// TIA Portal V17 export
// export: Created 2025-06-26T06:49:24.3780906Z, ExportSetting WithDefaults, DisplayName Totally Integrated Automation Portal, DisplayVersion V17 Update 8, DisplayName TIA Portal Openness, DisplayVersion V17 Update 8, DisplayName TIA Portal Version Control Interface, DisplayVersion V17, DisplayName STEP 7 Professional, DisplayVersion V17 Update 8, DisplayName STEP 7 Safety, DisplayVersion V17 Update 6, DisplayName WinCC Advanced, DisplayVersion V17 Update 8
DATA_BLOCK "HMI-Communication_DB"   // DB3
VERSION : 0.1
// stored: AutoNumber true, DBAccessibleFromOPCUA true, DBAccessibleFromWebserver true, InstanceOfName HMI-Communication, InstanceOfType FB
"HMI-Communication"
   // VAR
   //    StartRequest : Bool;
   //    StopRequest : Bool;
   //    HMI_Running : Bool;
   //    SkipPauseTime : Bool;
   //    EmergencyStopWaitTime : Bool;
   //    SkipEmergencyStopWait : Bool;
   //    CloseSafetyRelay : Bool;
   //    OpenSafetyRelay : Bool;
   //    HMI_Acknowledge_Error : Bool;
   //    BackToStandby_OilHeat { ExternalVisible := 'False'; ExternalWritable := 'False'} : Bool;
   //    BackToStandby_SourceFlowNotOK { ExternalVisible := 'False'; ExternalWritable := 'False'} : Bool;
   //    BackToStandby_SinkFlowNotOK : Bool;
   //    BackToStandby_SinkTemperatureNotOK : Bool;
   //    BackToStandby_SourceTemperatureNotOK : Bool;
   //    BackToStandby_PerformanceControlNotOK : Bool;
   //    ReturnValvesManualOverride : Bool;
   //    HBL_XV_02override : Bool;
   //    HBL_XV_03override : Bool;
   //    HBL_HV_860override : Bool;
   //    HBL_HV_861override : Bool;
   //    State_Text : String;
   //    BackToStandby_TriggerBit : Bool;
   //    BackToStandby_TriggerMemory : Bool;
   //    BackToStandby_TriggerInt : Int;
   //    BackToStandbyReason_Text : String;
   //    StopReason_TriggerBit : Bool;
   //    StopReason_TriggerMemory : Bool;
   //    StopReason_TriggerInt : Int;
   //    StopReason_Text : String;
   //    Progress_Text : Int;
   //    RegulationTarget : Int;
   //    RegulationTargetPrev : Int;
   //    HeatboosterSetpoint : Real;
   //    HeatboosterSetpointPrev : Real;
   //    EmergencyStopCountdown : Time_Of_Day;
   //    A1001 { ExternalAccessible := 'False'; ExternalVisible := 'False'; ExternalWritable := 'False'} : "fbHMIEvent";
   //    WinCCLink { ExternalAccessible := 'False'; ExternalVisible := 'False'; ExternalWritable := 'False'; S7_SetPoint := 'True'} : "fbHeartbeat";
   //    State2DwellTimeElapsed { S7_SetPoint := 'True'} : Time_Of_Day;
   //    State2DwellTime : Time_Of_Day;
   //    State3DwellTimeElapsed : Time_Of_Day;
   //    State3DwellTime : Time_Of_Day;
   //    State4DwellTimeElapsed : Time_Of_Day;
   //    State4DwellTime : Time_Of_Day;
   //    State5DwellTimeElapsed : Time_Of_Day;
   //    State5DwellTime : Time_Of_Day;
   //    State7DwellTimeElapsed : Time_Of_Day;
   //    State7DwellTime : Time_Of_Day;
   //    State2PauseTimeElapsed : Time_Of_Day;
   //    State2PauseTime : Time_Of_Day;
   //    PurgeControlPurgeTime : Time_Of_Day;
   //    PurgeControlSpinTime : Time_Of_Day;
   //    PerformanceControlStandbyTime : Time_Of_Day;
   //    PerformanceControlStandbyTimeElapsed : Time_Of_Day;
   //    FilterDryerOnTime : Time_Of_Day;
   //    FilterDryerOffTime : Time_Of_Day;
   //    OilRecoveryOnTime : Time_Of_Day;
   //    ProgressiveTimes : Array[0..3] of Time_Of_Day;
   //    ProgressiveTime : Time_Of_Day;
   //    ProgressiveManualTime : Time_Of_Day;
   //    HV640_OpenTime : Time_Of_Day;
   //    HV640_CloseTime : Time_Of_Day;
   //    HV670_OpenTime : Time_Of_Day;
   //    HV670_CloseTime : Time_Of_Day;
   //    HV852_OpenTime : Time_Of_Day;
   //    HV852_CloseTime : Time_Of_Day;
   //    HV861_OpenTime : Time_Of_Day;
   //    HV861_CloseTime : Time_Of_Day;
   //    State2DwellSync { ExternalAccessible := 'False'; ExternalVisible := 'False'; ExternalWritable := 'False'} : "fbWinCCTime";
   //    State3DwellSync { ExternalAccessible := 'False'; ExternalVisible := 'False'; ExternalWritable := 'False'; S7_SetPoint := 'True'} : "fbWinCCTime";
   //    State4DwellSync { ExternalAccessible := 'False'; ExternalVisible := 'False'; ExternalWritable := 'False'; S7_SetPoint := 'True'} : "fbWinCCTime";
   //    State5DwellSync { ExternalAccessible := 'False'; ExternalVisible := 'False'; ExternalWritable := 'False'; S7_SetPoint := 'True'} : "fbWinCCTime";
   //    State7DwellSync { ExternalAccessible := 'False'; ExternalVisible := 'False'; ExternalWritable := 'False'; S7_SetPoint := 'True'} : "fbWinCCTime";
   //    State2PauseSync { ExternalAccessible := 'False'; ExternalVisible := 'False'; ExternalWritable := 'False'; S7_SetPoint := 'True'} : "fbWinCCTime";
   //    PurgeControlPurgeSync { ExternalAccessible := 'False'; ExternalVisible := 'False'; ExternalWritable := 'False'; S7_SetPoint := 'True'} : "fbWinCCTime";
   //    PurgeControlSpinSync { ExternalAccessible := 'False'; ExternalVisible := 'False'; ExternalWritable := 'False'; S7_SetPoint := 'True'} : "fbWinCCTime";
   //    ProgressiveTime0Sync { ExternalAccessible := 'False'; ExternalVisible := 'False'; ExternalWritable := 'False'; S7_SetPoint := 'True'} : "fbWinCCTime";
   //    ProgressiveTime1Sync { ExternalAccessible := 'False'; ExternalVisible := 'False'; ExternalWritable := 'False'; S7_SetPoint := 'True'} : "fbWinCCTime";
   //    ProgressiveTime2Sync { ExternalAccessible := 'False'; ExternalVisible := 'False'; ExternalWritable := 'False'; S7_SetPoint := 'True'} : "fbWinCCTime";
   //    ProgressiveTime3Sync { ExternalAccessible := 'False'; ExternalVisible := 'False'; ExternalWritable := 'False'; S7_SetPoint := 'True'} : "fbWinCCTime";
   //    ProgressiveManualTimeSync { ExternalAccessible := 'False'; ExternalVisible := 'False'; ExternalWritable := 'False'; S7_SetPoint := 'True'} : "fbWinCCTime";
   //    PerformanceControlStandbySync { ExternalAccessible := 'False'; ExternalVisible := 'False'; ExternalWritable := 'False'; S7_SetPoint := 'True'} : "fbWinCCTime";
   //    FilterDryerOnTimeSync { S7_SetPoint := 'True'} : "fbWinCCTime";
   //    FilterDryerOffTimeSync { S7_SetPoint := 'True'} : "fbWinCCTime";
   //    OilRecoveryOnTimeSync { S7_SetPoint := 'True'} : "fbWinCCTime";
   //    HV640_OpenTimeSync { S7_SetPoint := 'True'} : "fbWinCCTime";
   //    HV640_CloseTimeSync { S7_SetPoint := 'True'} : "fbWinCCTime";
   //    HV670_OpenTimeSync { S7_SetPoint := 'True'} : "fbWinCCTime";
   //    HV670_CloseTimeSync { S7_SetPoint := 'True'} : "fbWinCCTime";
   //    HV852_OpenTimeSync { S7_SetPoint := 'True'} : "fbWinCCTime";
   //    HV852_CloseTimeSync { S7_SetPoint := 'True'} : "fbWinCCTime";
   //    HV861_OpenTimeSync { S7_SetPoint := 'True'} : "fbWinCCTime";
   //    HV861_CloseTimeSync { S7_SetPoint := 'True'} : "fbWinCCTime";
   // END_VAR
BEGIN
END_DATA_BLOCK
